(*	Struktura zawierające dane tylko tego elementu	*)
TYPE ST_Component_HMI :
STRUCT
	bZmiennaComponentHMI	: BOOL;

END_STRUCT
END_TYPE

(* stored: Version 1.1.0.1, ProductVersion 3.1.4024.15
   DUT ST_Component_HMI: Id {f58608a4-5954-4d37-86b7-4ce6ca0fa504} *)
